(* CoDeSys 2.3.9.62 project: CruceMoviles.pro *)
(* Libraries: Standard.lib 2.6.14 11:37:46 *)

(* Global variable list: Global_Variables *)
VAR_GLOBAL

      (*Entradas*)
      M1:BOOL;
      M2:BOOL;

	A1:BOOL;
	B1:BOOL;
       C1: BOOL;
       D1:BOOL;

	A2:BOOL;
	B2:BOOL;
      C2: BOOL;
       D2:BOOL;

       (* Salidas *)
	MOTOR_BA1:BOOL;
	MOTOR_FO1:BOOL;

       MOTOR_BA2:BOOL;
	MOTOR_FO2:BOOL;

      Carga1:BOOL;
      Carga2:BOOL;


      (* Variables del simulador *)
	Vel:INT:=1;
	Vel2:INT:=1;


END_VAR

(* POU PLC_PRG, ST *)
PROGRAM PLC_PRG
VAR
END_VAR
SimVehiculo;
SimVehiculo2;
Automatismo;
END_PROGRAM

(* POU SimVehiculo, ST *)
PROGRAM SimVehiculo
VAR
	PosX: INT;
END_VAR
A1:=FALSE;
B1:=FALSE;
C1:=FALSE;
D1:=FALSE;


IF MOTOR_FO1=TRUE THEN

     PosX:=PosX+Vel;

END_IF

IF MOTOR_BA1=TRUE THEN

     PosX:=PosX-Vel;

END_IF


IF PosX<=0 THEN
   A1:=TRUE;
END_IF

IF PosX>=129 AND   PosX<=199 THEN
   B1:=TRUE;
END_IF

IF PosX>=220 AND   PosX<=288 THEN
   C1:=TRUE;
END_IF

IF PosX>=438 THEN
  D1:=TRUE;
END_IF
END_PROGRAM

(* POU SimVehiculo2, ST *)
PROGRAM SimVehiculo2
VAR
	PosY2: INT;
END_VAR
A2:=FALSE;
B2:=FALSE;
C2:=FALSE;
D2:=FALSE;


IF MOTOR_FO2=TRUE THEN

     PosY2:=PosY2-Vel2;

END_IF

IF MOTOR_BA2=TRUE THEN

     PosY2:=PosY2+Vel2;

END_IF


IF PosY2>=0 THEN
   A2:=TRUE;
END_IF

IF PosY2<=-70 AND PosY2>=-142 THEN
  B2:=TRUE;
END_IF

IF PosY2<=-151 AND PosY2>=-220 THEN
  C2:=TRUE;
END_IF

IF PosY2<=-302  THEN
  D2:=TRUE;
END_IF
END_PROGRAM

(* POU Automatismo, LD *)
PROGRAM Automatismo
VAR

	Control1: ControlVehiculo;
	Control2: ControlVehiculo;
	OcupadoS2: BOOL;
	OcupadoS1: BOOL;
END_VAR
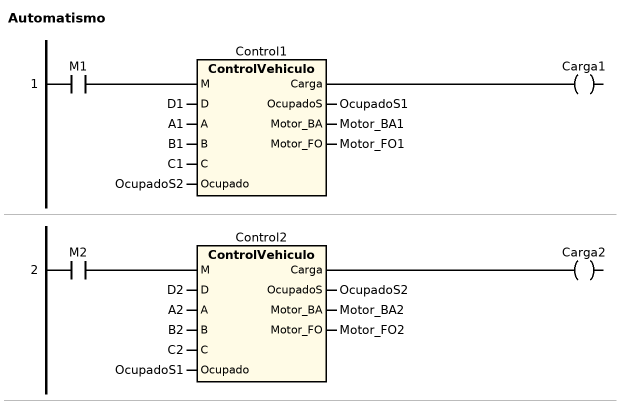
_LD_ (* Ladder Diagram *)
NETWORK 1
	[M1] - Control1:ControlVehiculo(M: *, D: D1, A: A1, B: B1, C: C1, Ocupado: OcupadoS2, OcupadoS => OcupadoS1, Motor_BA => Motor_BA1, Motor_FO => Motor_FO1) --- (Carga1)
NETWORK 2
	[M2] - Control2:ControlVehiculo(M: *, D: D2, A: A2, B: B2, C: C2, Ocupado: OcupadoS1, OcupadoS => OcupadoS2, Motor_BA => Motor_BA2, Motor_FO => Motor_FO2) --- (Carga2)
_END_LD_
(* the same logic as Structured Text *)
(* Network 1 *)
Control1(M := M1, D := D1, A := A1, B := B1, C := C1, Ocupado := OcupadoS2);
OcupadoS1 := Control1.OcupadoS;
Motor_BA1 := Control1.Motor_BA;
Motor_FO1 := Control1.Motor_FO;
Carga1 := Control1.Carga;
(* Network 2 *)
Control2(M := M2, D := D2, A := A2, B := B2, C := C2, Ocupado := OcupadoS1);
OcupadoS2 := Control2.OcupadoS;
Motor_BA2 := Control2.Motor_BA;
Motor_FO2 := Control2.Motor_FO;
Carga2 := Control2.Carga;
END_PROGRAM

(* POU ControlVehiculo, LD *)
FUNCTION_BLOCK ControlVehiculo
VAR_INPUT
	M: BOOL;
	D:BOOL;
	A: BOOL;
	B: BOOL;
	C:BOOL;
	Ocupado:BOOL;
END_VAR
VAR_OUTPUT
	Carga:BOOL;
	OcupadoS:BOOL;
	Motor_BA:BOOL;
	Motor_FO:BOOL;
END_VAR
VAR
	TCarga:TON;
	Contador: CTU;
	FinConta: BOOL;
	E1:BOOL;
	E2:BOOL;
	E3:BOOL;
	E4:BOOL;
	E5:BOOL;
	E6:BOOL;
	E7:BOOL;
	E8:BOOL;
	E9:BOOL;
	E10:BOOL;
	E11:BOOL;
	E12:BOOL;
END_VAR
VAR (* helpers for the ST form of the networks *)
	_p1 : BOOL;
	_p2 : BOOL;
	_p3 : BOOL;
	_p4 : BOOL;
	_p5 : BOOL;
	_p6 : BOOL;
	_p7 : BOOL;
	_p8 : BOOL;
	_p9 : BOOL;
	_p10 : BOOL;
	_p11 : BOOL;
	_p12 : BOOL;
	_p13 : BOOL;
	_p14 : BOOL;
	_p15 : BOOL;
END_VAR
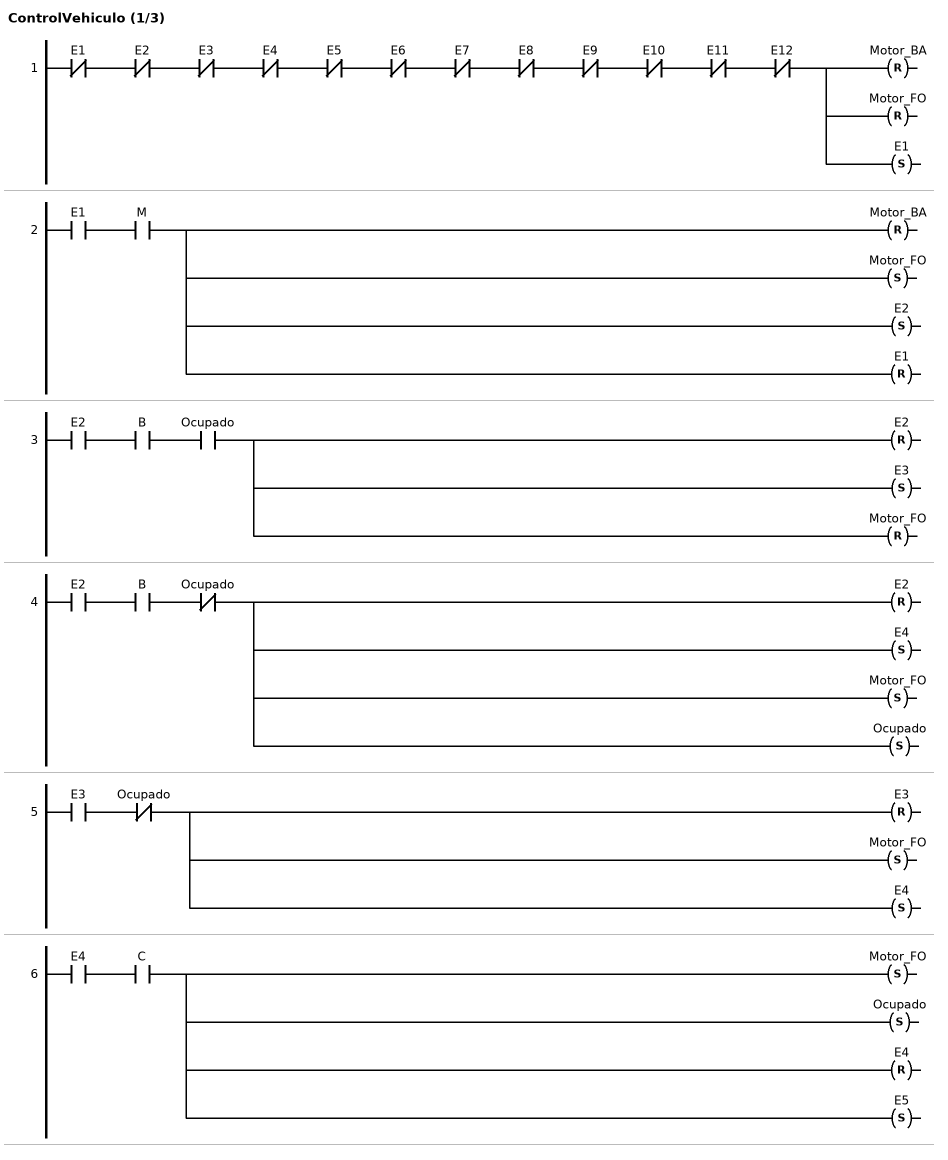
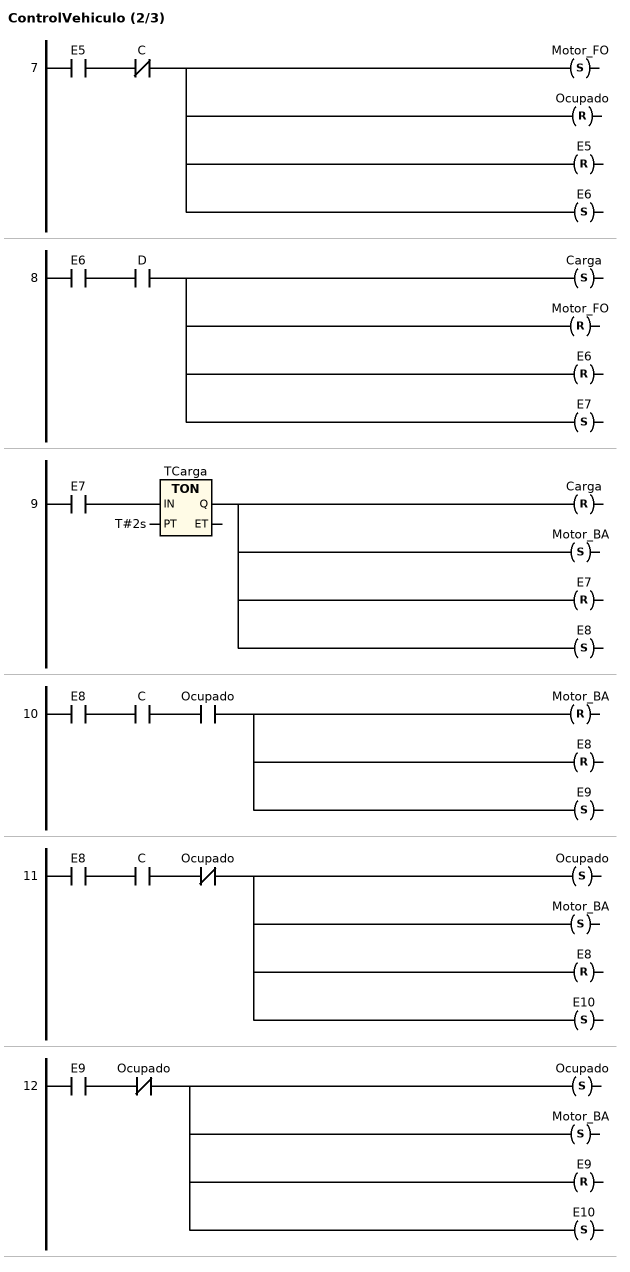
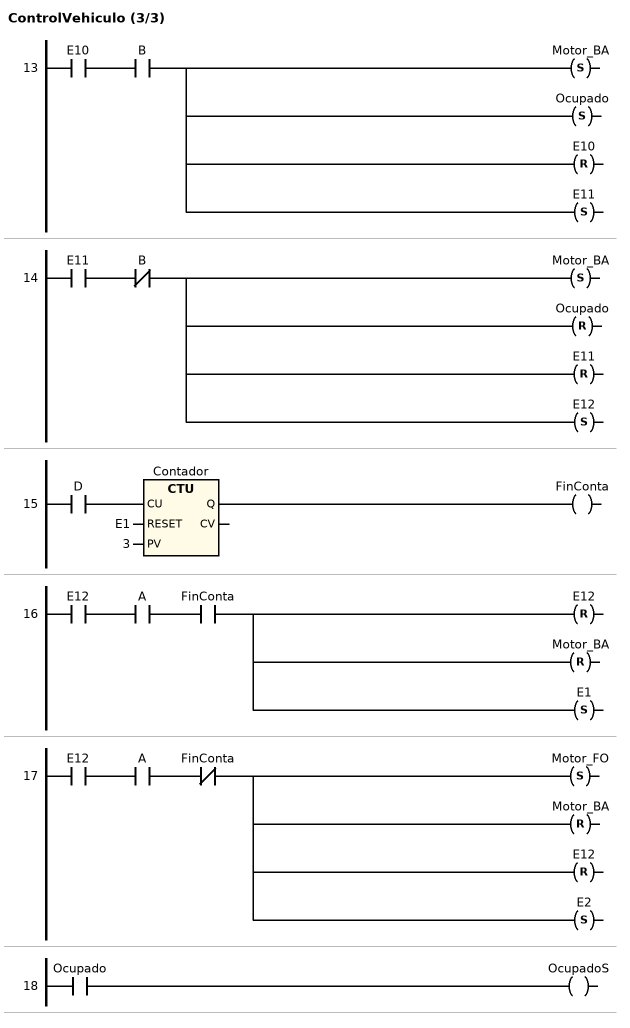
_LD_ (* Ladder Diagram *)
NETWORK 1
	[/E1] - [/E2] - [/E3] - [/E4] - [/E5] - [/E6] - [/E7] - [/E8] - [/E9] - [/E10] - [/E11] - [/E12] --- (R Motor_BA) (R Motor_FO) (S E1)
NETWORK 2
	[E1] - [M] --- (R Motor_BA) (S Motor_FO) (S E2) (R E1)
NETWORK 3
	[E2] - [B] - [Ocupado] --- (R E2) (S E3) (R Motor_FO)
NETWORK 4
	[E2] - [B] - [/Ocupado] --- (R E2) (S E4) (S Motor_FO) (S Ocupado)
NETWORK 5
	[E3] - [/Ocupado] --- (R E3) (S Motor_FO) (S E4)
NETWORK 6
	[E4] - [C] --- (S Motor_FO) (S Ocupado) (R E4) (S E5)
NETWORK 7
	[E5] - [/C] --- (S Motor_FO) (R Ocupado) (R E5) (S E6)
NETWORK 8
	[E6] - [D] --- (S Carga) (R Motor_FO) (R E6) (S E7)
NETWORK 9
	[E7] - TCarga:TON(IN: *, PT: T#2s) --- (R Carga) (S Motor_BA) (R E7) (S E8)
NETWORK 10
	[E8] - [C] - [Ocupado] --- (R Motor_BA) (R E8) (S E9)
NETWORK 11
	[E8] - [C] - [/Ocupado] --- (S Ocupado) (S Motor_BA) (R E8) (S E10)
NETWORK 12
	[E9] - [/Ocupado] --- (S Ocupado) (S Motor_BA) (R E9) (S E10)
NETWORK 13
	[E10] - [B] --- (S Motor_BA) (S Ocupado) (R E10) (S E11)
NETWORK 14
	[E11] - [/B] --- (S Motor_BA) (R Ocupado) (R E11) (S E12)
NETWORK 15
	[D] - Contador:CTU(CU: *, RESET: E1, PV: 3) --- (FinConta)
NETWORK 16
	[E12] - [A] - [FinConta] --- (R E12) (R Motor_BA) (S E1)
NETWORK 17
	[E12] - [A] - [/FinConta] --- (S Motor_FO) (R Motor_BA) (R E12) (S E2)
NETWORK 18
	[Ocupado] --- (OcupadoS)
_END_LD_
(* the same logic as Structured Text *)
(* Network 1 *)
_p1 := NOT E1 AND NOT E2 AND NOT E3 AND NOT E4 AND NOT E5 AND NOT E6 AND NOT E7 AND NOT E8 AND NOT E9 AND NOT E10 AND NOT E11 AND NOT E12;
IF _p1 THEN Motor_BA := FALSE; Motor_FO := FALSE; E1 := TRUE; END_IF;
(* Network 2 *)
_p2 := E1 AND M;
IF _p2 THEN Motor_BA := FALSE; Motor_FO := TRUE; E2 := TRUE; E1 := FALSE; END_IF;
(* Network 3 *)
_p3 := E2 AND B AND Ocupado;
IF _p3 THEN E2 := FALSE; E3 := TRUE; Motor_FO := FALSE; END_IF;
(* Network 4 *)
_p4 := E2 AND B AND NOT Ocupado;
IF _p4 THEN E2 := FALSE; E4 := TRUE; Motor_FO := TRUE; Ocupado := TRUE; END_IF;
(* Network 5 *)
_p5 := E3 AND NOT Ocupado;
IF _p5 THEN E3 := FALSE; Motor_FO := TRUE; E4 := TRUE; END_IF;
(* Network 6 *)
_p6 := E4 AND C;
IF _p6 THEN Motor_FO := TRUE; Ocupado := TRUE; E4 := FALSE; E5 := TRUE; END_IF;
(* Network 7 *)
_p7 := E5 AND NOT C;
IF _p7 THEN Motor_FO := TRUE; Ocupado := FALSE; E5 := FALSE; E6 := TRUE; END_IF;
(* Network 8 *)
_p8 := E6 AND D;
IF _p8 THEN Carga := TRUE; Motor_FO := FALSE; E6 := FALSE; E7 := TRUE; END_IF;
(* Network 9 *)
TCarga(IN := E7, PT := T#2s);
IF TCarga.Q THEN Carga := FALSE; Motor_BA := TRUE; E7 := FALSE; E8 := TRUE; END_IF;
(* Network 10 *)
_p9 := E8 AND C AND Ocupado;
IF _p9 THEN Motor_BA := FALSE; E8 := FALSE; E9 := TRUE; END_IF;
(* Network 11 *)
_p10 := E8 AND C AND NOT Ocupado;
IF _p10 THEN Ocupado := TRUE; Motor_BA := TRUE; E8 := FALSE; E10 := TRUE; END_IF;
(* Network 12 *)
_p11 := E9 AND NOT Ocupado;
IF _p11 THEN Ocupado := TRUE; Motor_BA := TRUE; E9 := FALSE; E10 := TRUE; END_IF;
(* Network 13 *)
_p12 := E10 AND B;
IF _p12 THEN Motor_BA := TRUE; Ocupado := TRUE; E10 := FALSE; E11 := TRUE; END_IF;
(* Network 14 *)
_p13 := E11 AND NOT B;
IF _p13 THEN Motor_BA := TRUE; Ocupado := FALSE; E11 := FALSE; E12 := TRUE; END_IF;
(* Network 15 *)
Contador(CU := D, RESET := E1, PV := 3);
FinConta := Contador.Q;
(* Network 16 *)
_p14 := E12 AND A AND FinConta;
IF _p14 THEN E12 := FALSE; Motor_BA := FALSE; E1 := TRUE; END_IF;
(* Network 17 *)
_p15 := E12 AND A AND NOT FinConta;
IF _p15 THEN Motor_FO := TRUE; Motor_BA := FALSE; E12 := FALSE; E2 := TRUE; END_IF;
(* Network 18 *)
OcupadoS := Ocupado;
END_FUNCTION_BLOCK

(* Visualisation Vehiculo
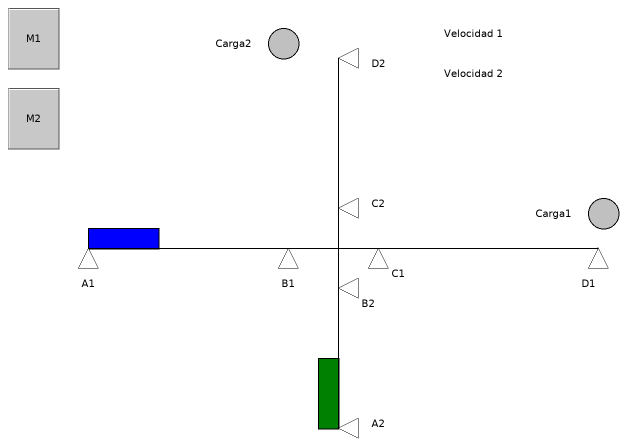
rectangle at (120,230)-(191,251): x offset SimVehiculo.PosX
polygon at (110,250)-(130,270): alarm colour if .A1
polygon at (620,250)-(640,270): alarm colour if .D1
button at (40,10)-(91,71): text "M1"; taps M1
rectangle at (350,360)-(371,431): y offset SimVehiculo2.PosY2
polygon at (370,420)-(390,440): alarm colour if .A2
rectangle at (450,20)-(561,51): text "Velocidad 1"
rectangle at (450,60)-(561,91): text "Velocidad 2"
polygon at (370,50)-(390,70): alarm colour if .D2
polygon at (310,250)-(330,270): alarm colour if .B1
polygon at (400,250)-(420,270): alarm colour if .C1
polygon at (370,280)-(390,300): alarm colour if .B2
polygon at (370,200)-(390,220): alarm colour if .C2
ellipse at (620,200)-(651,231): alarm colour if Carga1
rectangle at (530,200)-(641,231): text "Carga1"
ellipse at (300,30)-(331,61): alarm colour if Carga2
rectangle at (210,30)-(321,61): text "Carga2"
rectangle at (100,270)-(141,301): text "A1"
rectangle at (300,270)-(341,301): text "B1"
rectangle at (410,260)-(451,291): text "C1"
rectangle at (600,270)-(641,301): text "D1"
rectangle at (390,410)-(431,441): text "A2"
rectangle at (380,290)-(421,321): text "B2"
rectangle at (390,190)-(431,221): text "C2"
rectangle at (390,50)-(431,81): text "D2"
button at (40,90)-(91,151): text "M2"; taps M2
2 more shapes without text or variables
2 elements of other kinds (tables, trends, ...) not read
*)
